// TwinCAT 3 PLC project ContinousSync
// ProgramVersion: 3.1.4024.0
// libraries:
//   Tc2_MC2, * (Beckhoff Automation GmbH)
//   Tc2_MC2_FlyingSaw, * (Beckhoff Automation GmbH)
//   Tc2_Standard, * (Beckhoff Automation GmbH)
//   Tc2_System, * (Beckhoff Automation GmbH)
//   Tc3_Module, * (Beckhoff Automation GmbH)
//   VisuSymbols,3.5.10.0,System
// project tree:
//   / GlobalTextList.TcGTLO, PlcTask.TcTTO, Visualization Manager.TcVMO (not stored)
//   POUs/ MAIN.TcPOU, ContinousSync.TcPOU, States.TcDUT, SyncProgram.TcPOU
//   VISUs/ Visualization.TcVIS
// real-time tasks:
//   TASK PlcTask: cycle T#10ms, priority 20, ADS port 350
// motion (NC):
//   TASK NC-Task 1 SAF: cycle T#2ms, priority 4, ADS port 501
//   TASK NC-Task 1 SVB: cycle T#10ms, priority 8, ADS port 511
//   AXIS Axis 1 (id 1)
//     General: UnitName=Degree
//     OtherSettings: AllowMotionCmdToSlave=true
//     encoder EncType=19
//       EncPara: ScaleFactorNumerator=0.0054931640625, Offset=2370022.42, MaxCount=#xffffffff
//     drive DrvType=16
//       DrvPara: MaxCount=#xffffffff, DriveControlDWord=#x00020000
//         Analog: TorqueSetpointScale=10, ScaleFactorActTorque=0.1
//         TimeComp: TaskDelayCycles=1
//     controller CtrType=1
//       CtrPara: PriorControlFactor=1
//         PosDiffControl: Range=50
//         Observer: BandWidth=20
//   AXIS Axis 2 (id 2)
//     General: UnitName=Degree
//     OtherSettings: AllowMotionCmdToSlave=true
//     encoder EncType=19
//       EncPara: ScaleFactorNumerator=0.0054931640625, Offset=-4342912.4, MaxCount=#xffffffff
//     drive DrvType=16
//       DrvPara: MaxCount=#xffffffff, DriveControlDWord=#x00020000
//         Analog: TorqueSetpointScale=10, ScaleFactorActTorque=0.1
//         TimeComp: TaskDelayCycles=1
//     controller CtrType=1
//       CtrPara: PriorControlFactor=1
//         PosDiffControl: Range=50
//         Observer: BandWidth=20
// I/O:
//   DEVICE Device 2 (EtherCAT), AmsNetId 10.0.20.83.3.1
//     Drive 1 (Servo 9400 Highline TA CiA 402) [Servo 9400 Highline ECAT V3 TA CiA 402]
//     Drive 2 (Servo 9400 Highline TA CiA 402) [Servo 9400 Highline ECAT V2 TA CiA 402]
// variable links:
//   NC-Task 1 SAF/Axes/Axis 1 <-> Device 2 (EtherCAT)/Drive 1 (Servo 9400 Highline TA CiA 402)
//     Drive/Inputs/In/nState1 <-> Cylic Position Mode/Statusword
//     Drive/Inputs/In/nState2 <-> Cylic Position Mode/Statusword @bit 8
//     Drive/Inputs/In/nState4 @bit 1 <-> WcState/InputToggle
//     Drive/Inputs/In/nState4 <-> WcState/WcStateIn
//     Drive/Inputs/In/nState5 <-> Cylic Position Mode/Mode of Operation display
//     Drive/Outputs/Out/nCtrl1 <-> Cylic Position Mode_1/Controlword
//     Drive/Outputs/Out/nCtrl2 <-> Cylic Position Mode_1/Controlword @bit 8
//     Drive/Outputs/Out/nCtrl5 <-> Cylic Position Mode_1/Mode of Operation
//     Drive/Outputs/Out/nDataOut1 <-> Cylic Position Mode_1/Target position
//     Enc/Inputs/In/nDataIn1 <-> Cylic Position Mode/Position actual value (units)
//     Enc/Inputs/In/nState4 @bit 1 <-> WcState/InputToggle
//     Enc/Inputs/In/nState4 <-> WcState/WcStateIn
//   NC-Task 1 SAF/Axes/Axis 2 <-> Device 2 (EtherCAT)/Drive 2 (Servo 9400 Highline TA CiA 402)
//     Drive/Inputs/In/nState1 <-> Cylic Position Mode/Statusword
//     Drive/Inputs/In/nState2 <-> Cylic Position Mode/Statusword @bit 8
//     Drive/Inputs/In/nState4 @bit 1 <-> WcState/InputToggle
//     Drive/Inputs/In/nState4 <-> WcState/WcStateIn
//     Drive/Inputs/In/nState5 <-> Cylic Position Mode/Mode of Operation display
//     Drive/Outputs/Out/nCtrl1 <-> Cylic Position Mode_1/Controlword
//     Drive/Outputs/Out/nCtrl2 <-> Cylic Position Mode_1/Controlword @bit 8
//     Drive/Outputs/Out/nCtrl5 <-> Cylic Position Mode_1/Mode of Operation
//     Drive/Outputs/Out/nDataOut1 <-> Cylic Position Mode_1/Target position
//     Enc/Inputs/In/nDataIn1 <-> Cylic Position Mode/Position actual value (units)
//     Enc/Inputs/In/nState4 @bit 1 <-> WcState/InputToggle
//     Enc/Inputs/In/nState4 <-> WcState/WcStateIn
//   ContinousSync/ContinousSync Instance <-> NC-Task 1 SAF/Axes/Axis 1
//     PlcTask Inputs/SyncProgram.fbAxisSync.MasterAxis.NcToPlc <-> Outputs/ToPlc
//     PlcTask Outputs/SyncProgram.fbAxisSync.MasterAxis.PlcToNc <-> Inputs/FromPlc
//   ContinousSync/ContinousSync Instance <-> NC-Task 1 SAF/Axes/Axis 2
//     PlcTask Inputs/SyncProgram.fbAxisSync.SlaveAxis.NcToPlc <-> Outputs/ToPlc
//     PlcTask Outputs/SyncProgram.fbAxisSync.SlaveAxis.PlcToNc <-> Inputs/FromPlc

CONFIGURATION ContinousSync
    RESOURCE PLC ON TwinCAT3
        TASK PlcTask(INTERVAL := T#10ms, PRIORITY := 20);
        PROGRAM MAIN WITH PlcTask : MAIN;
    END_RESOURCE
END_CONFIGURATION

// ---- POUs/States.TcDUT
{attribute 'qualified_only'}
{attribute 'strict'}
TYPE States :
(
	CheckOnline := 0,
	StartMaster := 10,
	Synchronization := 20,
	ReadPosition := 30,
	ActivateFlyingSaw := 40,
	GearOut := 50,
	TempReset := 60,
	ErrorAndReset := 999,
	ReturnToPosition0 := 1000
);
END_TYPE

// ---- POUs/MAIN.TcPOU
PROGRAM MAIN
VAR
END_VAR

SyncProgram();

END_PROGRAM

// ---- POUs/SyncProgram.TcPOU
PROGRAM SyncProgram
VAR
	fbAxisSync : ContinousSync;
	bStartButton : BOOL;
	bStopButton : BOOL;
END_VAR

fbAxisSync.bStart := bStartButton;
fbAxisSync.bStop := bStopButton;

fbAxisSync();

END_PROGRAM

// ---- POUs/ContinousSync.TcPOU
FUNCTION_BLOCK ContinousSync
VAR_INPUT
	bStart : BOOL; //start the jogging of the master
	bStop : BOOL; //button to stop and reset the movement
END_VAR
VAR_OUTPUT
END_VAR
VAR
	iState : States;	
	
	rSyncPos : LREAL; //position where they sync
	
	fbGetSyncPos : R_TRIG; //we read the sync pos
	fbSyncTimer : TON; //timers that control when the sync and desync start
	fbDesyncTimer : TON;
	
	rActualMasterPos : LREAL; //the actual position of the master axis
	rActualSlavePos : LREAL; //the actual position of the slave axis	
	
	
	MasterAxis : AXIS_REF; //reference to the master and slave axis respectively
	SlaveAxis : AXIS_REF;
	
	PowerMaster : MC_Power; //power function blocks for the master and slave
	PowerSlave : MC_Power; 
	
	ResetMaster : MC_Reset; //reset function blocks for the master and slave
	ResetSlave : MC_Reset; 
	
	StopMaster : MC_Stop; //stop function blocks for the master and slave
	StopSlave : MC_Stop;

	JogMaster : MC_Jog; //function block to move the master
	
	FlyingSaw : MC_GearInPos; //function blocks for gearing in/out
	GearOut : MC_GearOut;
	
	MoveMaster : MC_MoveAbsolute;
	MoveSlave : MC_MoveAbsolute;
		
END_VAR

CASE iState OF
	States.CheckOnline: //check if the axes are turned on
		IF PowerMaster.Enable AND PowerSlave.Enable THEN
			iState := States.StartMaster;
		END_IF
		IF JogMaster.Error THEN
			iState := States.ErrorAndReset; //if an error occurs go to the error handling state
		END_IF
	States.StartMaster: //start the master if the button is pressed
		IF bStart THEN
			JogMaster(Axis := MasterAxis,JogForward := TRUE);
			iState := States.Synchronization;
		END_IF
	States.Synchronization: //start the sync process
		fbGetSyncPos(CLK := FALSE);
		fbSyncTimer.IN := TRUE;
		IF fbSyncTimer.Q THEN
			iState := States.ReadPosition;
		END_IF
		IF JogMaster.Error OR bStop THEN //incase an error or occurs or we stop it manually
			iState := States.ErrorAndReset;			
		END_IF
	States.ReadPosition: //write sync pos
		fbSyncTimer.IN := FALSE;
		fbGetSyncPos(CLK := TRUE); //we read the sync pos
		IF fbGetSyncPos.Q THEN
			rSyncPos := rActualMasterPos + 135.0;
			iState := States.ActivateFlyingSaw; 
		END_IF
		IF JogMaster.Error OR bStop THEN //incase an error or occurs or we stop it manually
			iState := States.ErrorAndReset;			
		END_IF
	States.ActivateFlyingSaw: //flying saw
		fbGetSyncPos(CLK := FALSE);
		FlyingSaw(Master := MasterAxis,Slave := SlaveAxis,MasterSyncPosition := rSyncPos,SlaveSyncPosition := rSyncPos,Execute := TRUE);
		fbDesyncTimer.IN := TRUE; //we start the desync timer
		IF fbDesyncTimer.Q THEN
			iState := States.GearOut;
		END_IF
		IF JogMaster.Error OR bStop THEN //incase an error or occurs or we stop it manually
			iState := States.ErrorAndReset;			
		END_IF
	States.GearOut: //Gear out and stop the slave
		fbDesyncTimer.IN := FALSE;
		StopSlave(Axis := SlaveAxis,Deceleration := 3000,Execute := TRUE);
		GearOut(Slave := SlaveAxis,Execute := TRUE);
		FlyingSaw(Master := MasterAxis,Slave := SlaveAxis,Execute := FALSE);
		IF StopSlave.Done THEN
			iState := States.TempReset; //reset all the blocks
		END_IF
		IF JogMaster.Error OR bStop THEN //incase an error or occurs or we stop it manually
			iState := States.ErrorAndReset;			
		END_IF
	States.TempReset: //reset gear out
		GearOut(Slave := SlaveAxis,Execute := FALSE);
		StopSlave(Axis := SlaveAxis,Execute := FALSE);
		iState := States.Synchronization;
	States.ErrorAndReset: //error and reset state
		GearOut(Slave := SlaveAxis,Execute := TRUE);
		StopSlave(Axis := SlaveAxis,Execute := TRUE);
		StopMaster(Axis := SlaveAxis,Execute := TRUE);
		fbSyncTimer.IN := FALSE;
		fbDesyncTimer.IN := FALSE;
		fbGetSyncPos(CLK := FALSE);
		JogMaster(Axis := MasterAxis,JogForward := FALSE);
		MoveMaster(Axis := MasterAxis,Execute := FALSE);
		MoveSlave(Axis := SlaveAXis,Execute := FALSE);
		IF JogMaster.Error OR MoveMaster.Error OR MoveSlave.Error THEN
			ResetMaster(Axis := MasterAxis,Execute := TRUE);
			ResetSlave(Axis := SlaveAxis,Execute := TRUE);
		ELSE
			iState := States.ReturnToPosition0; //return to the starting point
		END_IF

	States.ReturnToPosition0: //return to position 0
		GearOut(Slave := SlaveAxis,Execute := FALSE);
		StopSlave(Axis := SlaveAxis,Execute := FALSE);
		StopMaster(Axis := SlaveAxis,Execute := FALSE);
		ResetMaster(Axis := MasterAxis,Execute := FALSE);
		ResetSlave(Axis := SlaveAxis,Execute := FALSE);
		MoveMaster(Axis := MasterAxis,Position := 0,Velocity := 800,Execute := TRUE);
		MoveSlave(Axis := SlaveAxis,Position := 0,Velocity := 800,Execute := TRUE);
		IF MoveMaster.Done AND MoveSlave.Done THEN
			MoveMaster(Axis := MasterAxis,Execute := FALSE);
			MoveSlave(Axis := SlaveAxis,Execute := FALSE);
			iState := 10; //return to the start
		ELSIF MoveMaster.Error OR MoveSlave.Error THEN
			iState := States.ErrorAndReset;
		END_IF
						
END_CASE


PowerMaster(Axis := MasterAxis,Enable := TRUE,Enable_Positive := TRUE,Enable_Negative := TRUE);
PowerSlave(Axis := SlaveAxis,Enable := TRUE,Enable_Positive := TRUE,Enable_Negative := TRUE);

ResetMaster(Axis := MasterAxis);
ResetSlave(Axis := SlaveAxis);

StopMaster(Axis := MasterAxis);
StopSlave(Axis := SlaveAxis);

JogMaster(Axis := MasterAxis);

MoveMaster(Axis := MasterAxis);
MoveSlave(Axis := SlaveAXis);

fbSyncTimer(PT := T#4000MS);
fbDesyncTimer(PT := T#4000MS);

rActualMasterPos := MasterAxis.NcToPlc.ActPos;
rActualSlavePos := SlaveAxis.NcToPlc.ActPos;

END_FUNCTION_BLOCK

// ---- VISUs/Visualization.TcVIS
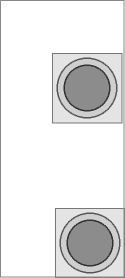
VISUALIZATION Visualization  // 125x278
    PushSwitchLed (52,53 70x70), variable: SyncProgram.bStartButton, behaviour: TAP, style: Switch-PushSwitchLed-Gray
    PushSwitchLed (55,208 70x70), variable: SyncProgram.bStopButton, behaviour: TAP, style: Switch-PushSwitchLed-Gray
END_VISUALIZATION
